ABB RobotStudio station: Proyecto_Final_B2.rspag

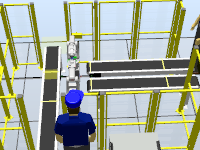
--- station ---
Station Station (saved by RobotStudio 20.4.9280.0)
Controller Controlador3, task T_ROB2: task frame (RAPID world) sits at (-70, -40, 300) mm, rotated rx 0 ry 0 rz -90 deg in the station
Controller Controlador3, task T_ROB1: task frame (RAPID world) sits at (-70, -40, 300) mm, rotated rx 0 ry 0 rz -90 deg in the station
Controller Controlador3
  mechanical unit ROB_1: IRB120_3_58__01, 6 joints, base frame (0, 0, 0) mm
  mechanical unit ROB_2: IRB120_3_58__01_2, 6 joints, base frame (820, 0, 0) mm, rotated rx 0 ry 0 rz 180 deg
Layout (positions relative to the parent item):
  - Conveyor_Cuchara [part]
  - Conveyor_Tenedor [part]
  - Conveyor_Caja [part]
  - Cuchara [part] at (-115.7, -210.79, 5) mm, rotated rx -173.75 ry 0 rz -55.83 deg
  - Tenedor [part] at (40.64, -627.66, 4.91) mm, rotated rx -174.81 ry 0 rz 176.86 deg
  - Logica_Conveyor_Cuchara [smart component]
      signals: DI Start6, DI Start10, DI Start12, DO Sensor_CucharaOK
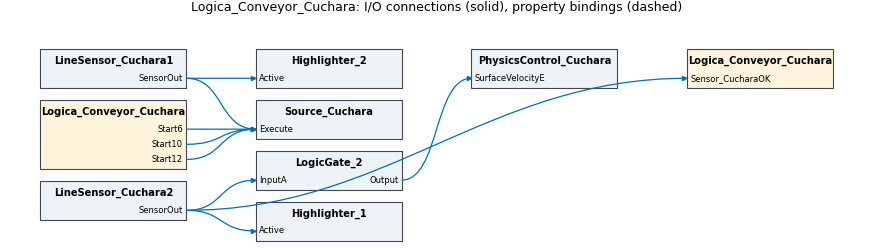
      connections:
        LineSensor_Cuchara1.SensorOut -> Source_Cuchara.Execute
        Logica_Conveyor_Cuchara.Start6 -> Source_Cuchara.Execute
        Logica_Conveyor_Cuchara.Start10 -> Source_Cuchara.Execute
        Logica_Conveyor_Cuchara.Start12 -> Source_Cuchara.Execute
        LineSensor_Cuchara2.SensorOut -> Logica_Conveyor_Cuchara.Sensor_CucharaOK
        LineSensor_Cuchara2.SensorOut -> LogicGate_2.InputA
        LogicGate_2.Output -> PhysicsControl_Cuchara.SurfaceVelocityEnabled
        LineSensor_Cuchara1.SensorOut -> Highlighter_2.Active
        LineSensor_Cuchara2.SensorOut -> Highlighter_1.Active
    - LineSensor_Cuchara1 [smart component, from Components\LineSensor.rslib]
        properties: Start=[1.5 -0.39 0.508]; End=[1.5 -0.11 0.508]; Radius=0.003; SensedPart=(none); SensedPoint=[0 0 0]
      - _sensorPart_ [part]
    - Source_Cuchara [smart component, from Components\Source.rslib]
        properties: Source=Cuchara; Copy=(none); Parent=(none); Position=[1.957 -0.257623 0.5035]; Orientation=[0.154636171726698 0.0188495559215388 0.00453785605518526]; Transient=true; PhysicsBehavior=3
    - LineSensor_Cuchara2 [smart component, from Components\LineSensor.rslib]
        properties: Start=[0.225 -0.39 0.508]; End=[0.225 -0.11 0.508]; Radius=0; SensedPart=(none); SensedPoint=[0.225 -0.212823776245117 0.508]
      - _sensorPart_ [part]
    - PhysicsControl_Cuchara [smart component, from Components\PhysicsControl.rslib]
        properties: Object=Conveyor_Cuchara; Behavior=1; SurfaceVelocity=0.3
    - LogicGate_2 [smart component, from Components\LogicGate.rslib]
        properties: Operator=NOT; Delay=0
    - Highlighter_1 [smart component, from Components\Highlighter.rslib]
        properties: Object=Pilot1; Color=[0 255 0]; Opacity=255
    - Highlighter_2 [smart component, from Components\Highlighter.rslib]
        properties: Object=Pilot2; Color=[0 255 0]; Opacity=255
  - Logica_Conveyor_Tenedor [smart component]
      signals: DI Start6, DI Start10, DI Start12, DO Sensor_TenedorOK
      connections:
        LineSensor_Tenedor.SensorOut -> Source_Tenedor.Execute
        Logica_Conveyor_Tenedor.Start6 -> Source_Tenedor.Execute
        Logica_Conveyor_Tenedor.Start10 -> Source_Tenedor.Execute
        Logica_Conveyor_Tenedor.Start12 -> Source_Tenedor.Execute
        LineSensor_3.SensorOut -> Logica_Conveyor_Tenedor.Sensor_TenedorOK
        LineSensor_3.SensorOut -> LogicGate.InputA
        LogicGate.Output -> PhysicsControl_Tenedor.SurfaceVelocityEnabled
        LineSensor_3.SensorOut -> Highlighter_3.Active
        LineSensor_Tenedor.SensorOut -> Highlighter_4.Active
    - LineSensor_Tenedor [smart component, from Components\LineSensor.rslib]
        properties: Start=[1.5 -0.8 0.508]; End=[1.5 -0.52 0.508]; Radius=0.003; SensedPart=(none); SensedPoint=[0 0 0]
      - _sensorPart_ [part]
    - Source_Tenedor [smart component, from Components\Source.rslib]
        properties: Source=Tenedor; Copy=(none); Parent=(none); Position=[1.957 -0.630695 0.505]; Orientation=[0 0 0]; Transient=true; PhysicsBehavior=3
    - LineSensor_3 [smart component, from Components\LineSensor.rslib]
        properties: Start=[0.228 -0.8 0.508]; End=[0.228 -0.52 0.508]; Radius=0; SensedPart=(none); SensedPoint=[0.227999984741211 -0.719083068847656 0.508]
      - _sensorPart_ [part]
    - PhysicsControl_Tenedor [smart component, from Components\PhysicsControl.rslib]
        properties: Object=Conveyor_Tenedor; Behavior=1; SurfaceVelocity=0.3
    - LogicGate [smart component, from Components\LogicGate.rslib]
        properties: Operator=NOT; Delay=0
    - Highlighter_3 [smart component, from Components\Highlighter.rslib]
        properties: Object=Pilot3; Color=[0 255 0]; Opacity=255
    - Highlighter_4 [smart component, from Components\Highlighter.rslib]
        properties: Object=Pilot4; Color=[0 255 0]; Opacity=255
  - Base_R_Tenedor [part] at (-70, -860, 0) mm
  - Base_R_Cuchara [part] at (-70, -40, 0) mm
  - Caja [part] at (-438.34, 1085.03, 1.58) mm, rotated rx 0 ry 0 rz -1.41 deg
  - Logica_Conveyor_Caja [smart component]
      signals: DI Start6, DI Start10, DI Start12, DO Sensor_CajaOK, DI Rutina
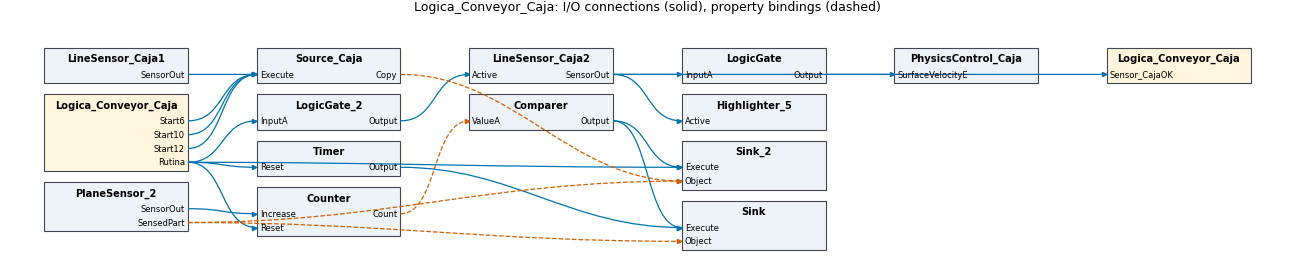
      connections:
        LineSensor_Caja1.SensorOut -> Source_Caja.Execute
        Logica_Conveyor_Caja.Start6 -> Source_Caja.Execute
        Logica_Conveyor_Caja.Start10 -> Source_Caja.Execute
        Logica_Conveyor_Caja.Start12 -> Source_Caja.Execute
        LineSensor_Caja2.SensorOut -> Logica_Conveyor_Caja.Sensor_CajaOK
        LineSensor_Caja2.SensorOut -> LogicGate.InputA
        LogicGate.Output -> PhysicsControl_Caja.SurfaceVelocityEnabled
        Logica_Conveyor_Caja.Rutina -> LogicGate_2.InputA
        LogicGate_2.Output -> LineSensor_Caja2.Active
        Logica_Conveyor_Caja.Rutina -> Sink_2.Execute
        LineSensor_Caja2.SensorOut -> Highlighter_5.Active
        PlaneSensor_2.SensorOut -> Counter.Increase
        Logica_Conveyor_Caja.Rutina -> Counter.Reset
        Comparer.Output -> Sink.Execute
        Comparer.Output -> Sink.Execute
        Timer.Output -> Sink.Execute
        Logica_Conveyor_Caja.Rutina -> Timer.Reset
        PlaneSensor_2.SensedPart => Sink.Object
        Source_Caja.Copy => Sink_2.Object
        Counter.Count => Comparer.ValueA
        PlaneSensor_2.SensedPart => Sink.Object
    - LineSensor_Caja1 [smart component, from Components\LineSensor.rslib]
        properties: Start=[-0.59 -1 0.515]; End=[-0.31 -1 0.515]; Radius=0.005; SensedPart=(none); SensedPoint=[0 0 0]
      - _sensorPart_ [part]
    - Source_Caja [smart component, from Components\Source.rslib]
        properties: Source=Caja2; Copy=(none); Parent=(none); Position=[-0.44646 -1.845404 0.503412]; Orientation=[0 0 0]; Transient=true; PhysicsBehavior=3
    - LineSensor_Caja2 [smart component, from Components\LineSensor.rslib]
        properties: Start=[-0.59 -0.35 0.515]; End=[-0.31 -0.35 0.515]; Radius=0.005; SensedPart=(none); SensedPoint=[-0.546462646484375 -0.35 0.515]
      - _sensorPart_ [part]
    - PhysicsControl_Caja [smart component, from Components\PhysicsControl.rslib]
        properties: Object=Conveyor_Caja; Behavior=1; SurfaceVelocity=0.3
    - LogicGate [smart component, from Components\LogicGate.rslib]
        properties: Operator=NOT; Delay=0
    - PlaneSensor_2 [smart component, from Components\PlaneSensor.rslib]
        properties: Origin=[-0.34 -0.555 0.5545]; Axis1=[-0.21 0 0]; Axis2=[0 0.22 0]; SensedPart=(none)
      - _sensorPart_ [part]
    - LogicGate_2 [smart component, from Components\LogicGate.rslib]
        properties: Operator=NOT; Delay=0
    - Highlighter_5 [smart component, from Components\Highlighter.rslib]
        properties: Object=Pilot5; Color=[0 255 0]; Opacity=255
    - Counter [smart component, from Components\Counter.rslib]
        properties: Count=3
    - Comparer [smart component, from Components\Comparer.rslib]
        properties: ValueA=3; Operator=>=; ValueB=4
    - Sink [smart component, from Components\Sink.rslib]
        properties: Object=(none)
    - Timer [smart component, from Components\Timer.rslib]
        properties: StartTime=10; Interval=10; Repeat=true; CurrentTime=13.728
  - IRB120_3_58__01 [mechanism, from Robots\IRB120_3_58_G_01.rslib] at (-70, -40, 300) mm, rotated rx 0 ry 0 rz -90 deg; joint values [0, 0, 0, 0, 0.5236, 0] (rad or m)
  - IRB120_3_58__01_2 [mechanism, from Robots\IRB120_3_58_G_01.rslib] at (-70, -860, 300) mm, rotated rx 0 ry 0 rz 90 deg; joint values [0, 0, 0, 0, 0.5236, 0] (rad or m)
  - Ventosa_tenedor [smart component, from Libraries\1217c23c-7d3e-48fb-b7d3-d1b2005a3c2bMi_Ventosa.rslib] at (-70, -495.65, 894) mm, rotated rx 180 ry 60 rz -90 deg
      connections:
        Ventosa_tenedor.DI_Coge_Objeto -> ?.Active
        ?.SensorOut -> Attacher.Execute
        Ventosa_tenedor.DI_Coge_Objeto -> LogicGate.InputA
        LogicGate.Output -> Detacher.Execute
        Ventosa_tenedor.DI_Coge_Objeto -> LineSensor.Active
        LineSensor.SensorOut -> Attacher.Execute
        LineSensor.SensedPart => Attacher.Child
        LineSensor.SensedPart => Detacher.Child
    - Attacher [smart component, from Components\Attacher.rslib]
        properties: Parent=Ventosa; Flange=0; Child=(none); Mount=false; Offset=[0 0 0]; Orientation=[0 0 0]
    - Detacher [smart component, from Components\Detacher.rslib]
        properties: Child=(none); KeepPosition=true
    - Ventosa [mechanism, from Libraries\1217c23c-7d3e-48fb-b7d3-d1b2005a3c2bMi_Ventosa.rslib] at (0, 0, 0) mm
    - LogicGate [smart component, from Components\LogicGate.rslib]
        properties: Operator=NOT; Delay=0
    - LineSensor [smart component, from Components\LineSensor.rslib]
        properties: Start=[5.20373137080643E-08 6.3539233263743E-08 0.0549999072719709]; End=[5.18797551862793E-08 6.35131238713171E-08 0.062499907271971]; Radius=0; SensedPart=(none); SensedPoint=[-0.419999938964844 -0.519800048828125 0.560922058105469]
      - _sensorPart_ [part]
    - Indicador [part, from Libraries\1217c23c-7d3e-48fb-b7d3-d1b2005a3c2bMi_Ventosa.rslib] at (-4.38, 0, 0) mm
  - Ventosa_cuchara [smart component, from Libraries\1217c23c-7d3e-48fb-b7d3-d1b2005a3c2bMi_Ventosa.rslib] at (-70, -404.35, 894) mm, rotated rx 180 ry 60 rz 90 deg
      connections:
        Ventosa_cuchara.DI_Coge_Objeto -> ?.Active
        ?.SensorOut -> Attacher.Execute
        Ventosa_cuchara.DI_Coge_Objeto -> LogicGate.InputA
        LogicGate.Output -> Detacher.Execute
        Ventosa_cuchara.DI_Coge_Objeto -> LineSensor.Active
        LineSensor.SensorOut -> Attacher.Execute
        LineSensor.SensedPart => Attacher.Child
        LineSensor.SensedPart => Detacher.Child
    - Attacher [smart component, from Components\Attacher.rslib]
        properties: Parent=Ventosa; Flange=0; Child=(none); Mount=false; Offset=[0 0 0]; Orientation=[0 0 0]
    - Detacher [smart component, from Components\Detacher.rslib]
        properties: Child=(none); KeepPosition=true
    - Ventosa [mechanism, from Libraries\1217c23c-7d3e-48fb-b7d3-d1b2005a3c2bMi_Ventosa.rslib] at (0, 0, 0) mm
    - LogicGate [smart component, from Components\LogicGate.rslib]
        properties: Operator=NOT; Delay=0
    - LineSensor [smart component, from Components\LineSensor.rslib]
        properties: Start=[0 0 0.055]; End=[-1.13103603149867E-08 -1.19271307830182E-08 0.0619999031141458]; Radius=0; SensedPart=(none); SensedPoint=[-0.419999969482422 -0.376149993896484 0.56155517578125]
      - _sensorPart_ [part]
    - Indicador [part, from Libraries\1217c23c-7d3e-48fb-b7d3-d1b2005a3c2bMi_Ventosa.rslib] at (-4.38, 0, 0) mm
  - Fence [graphiccomponentgroup]
    - Segment 1 [part]
    - Segment 2 [part]
    - Segment 3 [part]
    - Segment 4 [part]
    - Segment 5 [part]
  - Fence [graphiccomponentgroup]
    - Segment 1 [part]
    - Segment 2 [part]
    - Segment 3 [part]
    - Segment 4 [part]
    - Segment 5 [part]
  - Fence [graphiccomponentgroup]
    - Segment 1 [part]
    - Segment 2 [part]
    - Segment 3 [part]
    - Segment 4 [part]
    - Segment 5 [part]
    - Segment 6 [part]
  - IRC5_Control-Module [part, from Equipment\IRC5_Control-Module.rslib] at (800, -2180, 100) mm, rotated rx 90 ry 0 rz 0 deg
  - PlaneSensor [smart component, from Components\PlaneSensor.rslib]
      properties: Origin=[-0.7 0.32 0.3]; Axis1=[0.5 0 0]; Axis2=[0 0.5 0]; SensedPart=(none)
    - _sensorPart_ [part]
  - Sink [smart component, from Components\Sink.rslib]
      properties: Object=(none)
  - Man2 [part, from Libraries\b1fed280-7d32-4964-bca3-7f8177a599d8man2.rslib] at (2300, 0, 0) mm, rotated rx 0 ry 0 rz 180 deg
  - Man2_2 [part, from Libraries\b1fed280-7d32-4964-bca3-7f8177a599d8man2.rslib] at (-100, -2200, 0) mm, rotated rx 0 ry 0 rz 90 deg
  - Placa1 [part] at (200, -410, 400) mm
  - Placa3 [part] at (-200, -620, -50) mm
  - Placa2 [part]
  - Placa4 [part]
  - Placa5 [part]
  - Pilot5 [part]
  - Pilot1 [part]
  - Pilot2 [part]
  - Pilot4 [part]
  - Pilot3 [part]
  - Placa6 [part]
  - Pilot_r_tenedor [part] at (0, 14.72, 0) mm
  - Pilot_r_cuchara [part] at (0, -7.35, 0) mm
  - Highlighter_r_cuchara [smart component, from Components\Highlighter.rslib]
      properties: Object=Pilot_r_cuchara; Color=[0 255 0]; Opacity=255
  - Highlighter_r_tenedor [smart component, from Components\Highlighter.rslib]
      properties: Object=Pilot_r_tenedor; Color=[0 255 0]; Opacity=255
  - Caja2 [part] at (-14.34, -14695.99, 1.59) mm, rotated rx 0 ry 0 rz 5.75 deg
Attachment: Ventosa_tenedor is attached to IRB120_3_58__01_2 / Link6
Attachment: Ventosa_cuchara is attached to IRB120_3_58__01 / Link6
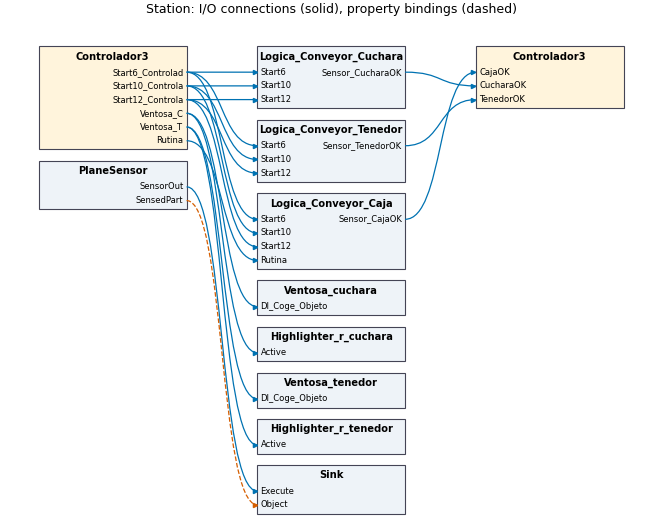
Station logic (signal -> signal, property => property):
  Controlador3.Start6_Controlador -> Logica_Conveyor_Caja.Start6
  Controlador3.Start10_Controlador -> Logica_Conveyor_Caja.Start10
  Controlador3.Start12_Controlador -> Logica_Conveyor_Caja.Start12
  Controlador3.Start6_Controlador -> Logica_Conveyor_Cuchara.Start6
  Controlador3.Start10_Controlador -> Logica_Conveyor_Cuchara.Start10
  Controlador3.Start12_Controlador -> Logica_Conveyor_Cuchara.Start12
  Controlador3.Start6_Controlador -> Logica_Conveyor_Tenedor.Start6
  Controlador3.Start10_Controlador -> Logica_Conveyor_Tenedor.Start10
  Controlador3.Start12_Controlador -> Logica_Conveyor_Tenedor.Start12
  Logica_Conveyor_Caja.Sensor_CajaOK -> Controlador3.CajaOK
  Logica_Conveyor_Cuchara.Sensor_CucharaOK -> Controlador3.CucharaOK
  Logica_Conveyor_Tenedor.Sensor_TenedorOK -> Controlador3.TenedorOK
  Controlador3.Ventosa_C -> Ventosa_cuchara.DI_Coge_Objeto
  Controlador3.Ventosa_T -> Ventosa_tenedor.DI_Coge_Objeto
  Controlador3.Rutina -> Logica_Conveyor_Caja.Rutina
  PlaneSensor.SensorOut -> Sink.Execute
  Controlador3.Ventosa_C -> Highlighter_r_cuchara.Active
  Controlador3.Ventosa_T -> Highlighter_r_tenedor.Active
  PlaneSensor.SensedPart => Sink.Object

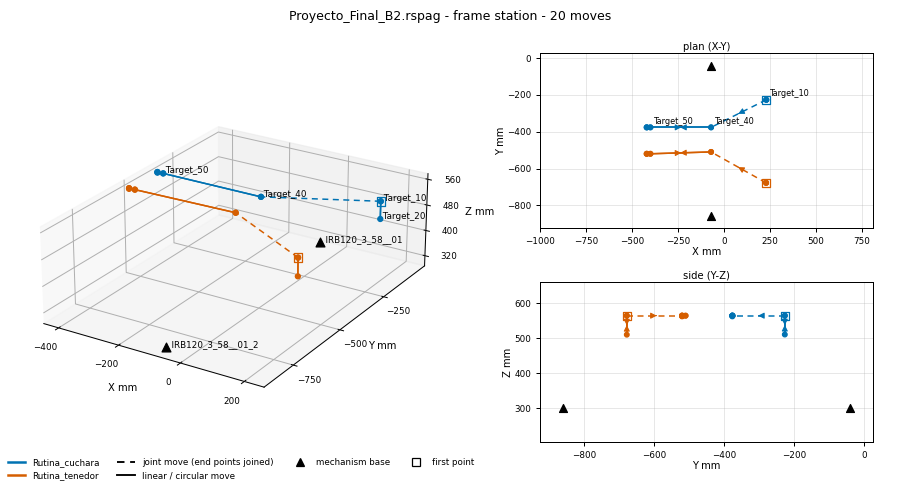
[picture p0: tool path of Proyecto_Final_B2.rspag in frame station, 20 of 20 moves have a stored position in this frame; points joined in program order, loops and branches not executed]
--- Backups/Controlador3/RAPID/TASK1/PROGMOD/CalibData.mod ---
MODULE CalibData
    PERS tooldata TCP_Ventosa:=[TRUE,[[0,0,60],[1,0,0,0]],[0.1,[0,0,1],[1,0,0,0],0,0,0]];
    TASK PERS wobjdata Workobject_1:=[FALSE,TRUE,"",[[210,270,200],[1,0,0,0]],[[0,0,0],[1,0,0,0]]];
    PERS tooldata Tooldata_1:=[TRUE,[[0,0,60],[1,0,0,0]],[0.1,[0,0,1],[1,0,0,0],0,0,0]];
ENDMODULE

--- Backups/Controlador3/RAPID/TASK1/PROGMOD/Module1.mod ---
MODULE Module1
    CONST robtarget Target_10:=[[-23.679995733,30.000024272,64.999939178],[0.000000004,0,1,0.000000007],[0,0,0,0],[9E+09,9E+09,9E+09,9E+09,9E+09,9E+09]];
    CONST robtarget Target_20:=[[-23.68,30,11.2],[0,0,1,0],[0,0,0,0],[9E+09,9E+09,9E+09,9E+09,9E+09,9E+09]];
    CONST robtarget Target_30:=[[-23.679995733,30.000024272,64.999939178],[0.000000004,0,1,0.000000007],[0,0,0,0],[9E+09,9E+09,9E+09,9E+09,9E+09,9E+09]];
    CONST robtarget Target_40:=[[126.149990693,-270.119999999,64.999933168],[0.000000011,0.486182918,0.873857065,0.000000019],[-1,0,0,0],[9E+09,9E+09,9E+09,9E+09,9E+09,9E+09]];
    CONST robtarget Target_50:=[[126.149993351,-600.000025877,64.999935931],[0.000000004,0.4861829,0.873857075,-0.000000015],[-1,-1,0,0],[9E+09,9E+09,9E+09,9E+09,9E+09,9E+09]];
    CONST robtarget Target_60:=[[126.15,-620,65],[0,0.707106781,0.707106781,0],[-1,-1,0,0],[9E+09,9E+09,9E+09,9E+09,9E+09,9E+09]];
    CONST robtarget Target_70:=[[126.15,-620,63],[0,0.707106781,0.707106781,0],[-1,-1,0,0],[9E+09,9E+09,9E+09,9E+09,9E+09,9E+09]];
    VAR num contador:=0;
    !***********************************************************
    !
    ! Módulo:  Module1
    !
    ! Descripción:
    !   <Introduzca la descripción aquí>
    !
    ! Autor: Admin
    !
    ! Versión: 1.0
    !
    !***********************************************************


    !***********************************************************
    !
    ! Procedimiento Main
    !
    !   Este es el punto de entrada de su programa
    !
    !***********************************************************
    !Declaración de variables de interrupción

    VAR intnum int_buttonStopDI;                           !intnum comando que identifica interrupcion de parada de emergencia.

    PROC main()
        !Añada aquí su código
        setDO Start6_Controlador,0;
        setDO Start10_Controlador,0;
        setDO Start12_Controlador,0;
        SetDO Ventosa_C,0;
        SetDO Rutina,0;
        ciclo_inicio_cuchara:
        IF cubiertos_6=high THEN
            IDelete int_buttonStopDI;                          !Cancela interrupcion, necesario cuando el ciclo se repite.
            CONNECT int_buttonStopDI WITH parada_emergencia;   !Se conecta la rutina TRAP con la interrupicion parada_emergencia
            iSignalDI Stop_button, 1, int_buttonStopDI;         !Se asocia buttonStop con la interrupcion parada_emergencia
            setDO Start6_Controlador,1;
            !setDO Start6_Controlador, 0;
            contador:=6;
            Rutina_cuchara;
            SetDO Rutina,1;
            WaitTime 1.5;
            SetDO Rutina,0;
        ELSEIF cubiertos_10=high THEN
            IDelete int_buttonStopDI;                          !Cancela interrupcion, necesario cuando el ciclo se repite.
            CONNECT int_buttonStopDI WITH parada_emergencia;   !Se conecta la rutina TRAP con la interrupicion parada_emergencia
            iSignalDI Stop_button, 1, int_buttonStopDI;         !Se asocia buttonStop con la interrupcion parada_emergencia
            setDO Start10_Controlador,1;
            !setDO Start10_Controlador, 0;
            contador:=10;
            Rutina_cuchara;
            SetDO Rutina,1;
            WaitTime 1.5;
            SetDO Rutina,0;
        ELSEIF cubiertos_12=high THEN
            IDelete int_buttonStopDI;                          !Cancela interrupcion, necesario cuando el ciclo se repite.
            CONNECT int_buttonStopDI WITH parada_emergencia;   !Se conecta la rutina TRAP con la interrupicion parada_emergencia
            iSignalDI Stop_button, 1, int_buttonStopDI;         !Se asocia buttonStop con la interrupcion parada_emergencia
            setDO Start12_Controlador,1;
            !setDO Start12_Controlador, 0;
            contador:=12;
            Rutina_cuchara;
            SetDO Rutina,1;
            WaitTime 1.5;
            SetDO Rutina,0;
        ELSE
            GOTO ciclo_inicio_cuchara;
        ENDIF
    ENDPROC
    PROC Rutina_cuchara()
        WHILE contador>0 DO
            WaitDI CajaOK,1;
            WaitDI CucharaOK,1;
            WaitDI TenedorOK,1;
            MoveJ Target_10,v600,z10,TCP_Ventosa\WObj:=Workobject_1;
            MoveL Target_20,v50,z1,TCP_Ventosa\WObj:=Workobject_1;
            SetDO Ventosa_C,1;
            WaitTime 1;
            MoveL Target_30,v150,z1,TCP_Ventosa\WObj:=Workobject_1;
            MoveJ Target_40,v600,z10,TCP_Ventosa\WObj:=Workobject_1;
            MoveL Target_50,v300,z1,TCP_Ventosa\WObj:=Workobject_1;
            MoveL Target_60,v300,z1,TCP_Ventosa\WObj:=Workobject_1;
            MoveL Target_70,v10,fine,Tooldata_1\WObj:=Workobject_1;
            SetDO Ventosa_C,0;
            WaitTime 1;
            MoveL Target_60,v300,z1,TCP_Ventosa\WObj:=Workobject_1;
            MoveL Target_50,v300,z1,TCP_Ventosa\WObj:=Workobject_1;
            MoveL Target_40,v300,z1,TCP_Ventosa\WObj:=Workobject_1;
            contador:=contador-1;
            IF contador=0 THEN
                IF cubiertos_6=high THEN
                   contador:=6;
                   SetDO Rutina,1;
                   WaitTime 1.5;
                   SetDO Rutina,0;
                ELSEIF cubiertos_10=high THEN
                   contador:=10;
                   SetDO Rutina,1;
                   WaitTime 1.5;
                   SetDO Rutina,0;
                ELSEIF cubiertos_12=high THEN
                   contador:=12;
                   SetDO Rutina,1;
                   WaitTime 1.5;
                   SetDO Rutina,0;
                ENDIF
            ENDIF
        ENDWHILE
    ENDPROC

    TRAP parada_emergencia                              !Interrupcion parada_emergencia
        StopMove;                                       !Detiene movimento de robot
        SetDO Rutina,0;
        !IF buttonStop=low THEN
        !    StartMove;
        !ELSE
        !    parada_emergencia:
        !ENDIF
        WHILE Stop_button = high DO                      !Mientras siga activo pulsador buttonStop, el programa seguirá detenido
        ENDWHILE
        StartMove;                                      !Si se desactiva pulsador buttonStop, el programa continua donde quedó.
    ENDTRAP
ENDMODULE

--- Backups/Controlador3/RAPID/TASK1/SYSMOD/LINKEDM.sys ---
%%%
  VERSION:1
  LANGUAGE:ENGLISH
%%%

MODULE LINKEDM (SYSMODULE)

! FOLLOWER
!     Name of electronically linked follower axis used by operator at teach pendent.
      PERS string l_f_axis_name{5}       :=  ["",  "", "", "", ""];

!     Name of the mechanical unit for follower axis.
      PERS string l_f_mecunt_n{5}  :=  ["", "", "", "", ""];

!     Linked follower axis number in the mechanical unit (first axis in mech. unit is number 1).
      PERS num l_f_axis_no{5}      :=  [0,          0,   0,  0,  0];

! MASTER
!     Name of the mechanical unit for linked master axis.
      PERS string l_m_mecunt_n{5} :=  ["", "", "", "", ""];

!     Linked master axis number in the mechanical unit (first axis in mech. unit is number 1).
!     See axis number table in documentation for different master mechanical units.
      PERS num l_m_axis_no{5}     :=  [0,  0,  0,  0,  0];

! POSITION OFFSET
!     The increase of the allowed offset position between the master and follower
!     positions, used when starting AUTO mode. As soon as the offset is decreased
!     the old configurated parameter is used.
!     Example: 3 => the configurated value of allowed offset is increased 3 times.
      PERS num offset_ratio{5}       :=  [10,  10,   10,  10,  10];

! SPEED RATIO
!     Speed_ratio used in AUTO and JOG modes [ very_slow   slow    normal    fast]
!     Value 1 = max allowed manual speed.
      CONST num speed_ratio {20}      := [0.01, 0.01, 0.01, 0.01, 0.01,
                                          0.05, 0.05, 0.05, 0.05, 0.05,
                                          0.20, 0.20, 0.20, 0.20, 0.20,
                                          1.00, 1.00, 1.00, 1.00, 1.00];

! STEP SIZE
!     Displacement position used in JOG mode for each activation of positive or
!     negative movement.                  [very_short    short   normal   long]
!     Unit degees or meter.
      CONST num displacement {20}     := [0.001, 0.001, 0.001, 0.001, 0.001,
                                          0.005, 0.005, 0.005, 0.005, 0.005,
                                          0.020, 0.020, 0.020, 0.020, 0.020,
                                          0.100, 0.100, 0.100, 0.100, 0.100];


!-------------------------------------------------------------
 PROC Linked_m ()
      Linked_m_exe ;
 ENDPROC
ENDMODULE

--- Backups/Controlador3/RAPID/TASK2/PROGMOD/CalibData.mod ---
MODULE CalibData
    PERS tooldata TCP_Ventosa:=[TRUE,[[0,0,60],[1,0,0,0]],[0.1,[0,0,1],[1,0,0,0],0,0,0]];
    TASK PERS wobjdata Workobject_2:=[FALSE,TRUE,"",[[620,270,200],[1,0,0,0]],[[0,0,0],[1,0,0,0]]];
ENDMODULE

--- Backups/Controlador3/RAPID/TASK2/PROGMOD/Module1.mod ---
MODULE Module1
    CONST robtarget Target_10:=[[17.680006378,29.000003785,64.999943406],[-0.000000006,1,0,0.000000004],[-1,0,-1,0],[9E+09,9E+09,9E+09,9E+09,9E+09,9E+09]];
    CONST robtarget Target_20:=[[17.68,29,10.7],[0,1,0,0],[-1,-1,-1,0],[9E+09,9E+09,9E+09,9E+09,9E+09,9E+09]];
    CONST robtarget Target_30:=[[17.680006378,29.000003785,64.999943406],[-0.000000006,1,0,0.000000004],[-1,0,-1,0],[9E+09,9E+09,9E+09,9E+09,9E+09,9E+09]];
    CONST robtarget Target_40:=[[-150.200005115,-270.140000008,64.999941394],[-0.000000007,0.871855665,0.489762902,0.000000004],[0,0,-1,0],[9E+09,9E+09,9E+09,9E+09,9E+09,9E+09]];
    CONST robtarget Target_50:=[[-140.200013899,-600.000004341,64.999949592],[0.000000013,0.871855673,0.489762887,0.000000004],[0,-1,-1,0],[9E+09,9E+09,9E+09,9E+09,9E+09,9E+09]];
    CONST robtarget Target_60:=[[-140.2,-620,65],[0,0.707106781,0.707106781,0],[0,-1,-1,0],[9E+09,9E+09,9E+09,9E+09,9E+09,9E+09]];
    CONST robtarget Target_70:=[[-140.2,-620,63],[0,0.707106781,0.707106781,0],[0,0,-1,0],[9E+09,9E+09,9E+09,9E+09,9E+09,9E+09]];
    VAR num contador:=0;
    !***********************************************************
    !
    ! Módulo:  Module1
    !
    ! Descripción:
    !   <Introduzca la descripción aquí>
    !
    ! Autor: Admin
    !
    ! Versión: 1.0
    !
    !***********************************************************


    !***********************************************************
    !
    ! Procedimiento Main
    !
    !   Este es el punto de entrada de su programa
    !
    !***********************************************************
    !Declaración de variables de interrupción

    VAR intnum int_buttonStopDI;                           !intnum comando que identifica interrupcion de parada de emergencia.

    PROC main()
        !Añada aquí su código
        setDO Start6_Controlador,0;
        setDO Start10_Controlador,0;
        setDO Start12_Controlador,0;
        SetDO Rutina,0;
        SetDO Ventosa_T,0;
        ciclo_inicio_tenedor:
        IF cubiertos_6=high THEN
            IDelete int_buttonStopDI;                          !Cancela interrupcion, necesario cuando el ciclo se repite.
            CONNECT int_buttonStopDI WITH parada_emergencia;   !Se conecta la rutina TRAP con la interrupicion parada_emergencia
            iSignalDI Stop_button, 1, int_buttonStopDI;         !Se asocia buttonStop con la interrupcion parada_emergencia
            setDO Start6_Controlador,1;
            !setDO Start6_Controlador, 0;
            contador:=6;
            Rutina_tenedor;
            SetDO Rutina,1;
            WaitTime 1.5;
            SetDO Rutina,0;
        ELSEIF cubiertos_10=high THEN
            IDelete int_buttonStopDI;                          !Cancela interrupcion, necesario cuando el ciclo se repite.
            CONNECT int_buttonStopDI WITH parada_emergencia;   !Se conecta la rutina TRAP con la interrupicion parada_emergencia
            iSignalDI Stop_button, 1, int_buttonStopDI;         !Se asocia buttonStop con la interrupcion parada_emergencia
            setDO Start10_Controlador,1;
            !setDO Start10_Controlador, 0;
            contador:=10;
            Rutina_tenedor;
            SetDO Rutina,1;
            WaitTime 1.5;
            SetDO Rutina,0;
        ELSEIF cubiertos_12=high THEN
            IDelete int_buttonStopDI;                          !Cancela interrupcion, necesario cuando el ciclo se repite.
            CONNECT int_buttonStopDI WITH parada_emergencia;   !Se conecta la rutina TRAP con la interrupicion parada_emergencia
            iSignalDI Stop_button, 1, int_buttonStopDI;         !Se asocia buttonStop con la interrupcion parada_emergencia
            setDO Start12_Controlador,1;
            !setDO Start12_Controlador, 0;
            contador:=12;
            Rutina_tenedor;
            SetDO Rutina,1;
            WaitTime 1.5;
            SetDO Rutina,0;
        ELSE
            GOTO ciclo_inicio_tenedor;
        ENDIF
    ENDPROC
    PROC Rutina_tenedor()
        WHILE contador>0 DO
            WaitDI CajaOK,1;
            WaitDI CucharaOK,1;
            WaitDI TenedorOK,1;
            MoveJ Target_10,v600,z10,TCP_Ventosa\WObj:=Workobject_2;
            MoveL Target_20,v50,z1,TCP_Ventosa\WObj:=Workobject_2;
            SetDO Ventosa_T,1;
            WaitTime 1;
            MoveL Target_30,v150,z1,TCP_Ventosa\WObj:=Workobject_2;
            MoveJ Target_40,v600,z10,TCP_Ventosa\WObj:=Workobject_2;
            MoveL Target_50,v300,z1,TCP_Ventosa\WObj:=Workobject_2;
            MoveL Target_60,v300,z1,TCP_Ventosa\WObj:=Workobject_2;
            MoveL Target_70,v10,fine,TCP_Ventosa\WObj:=Workobject_2;
            SetDO Ventosa_T,0;
            WaitTime 1;
            MoveL Target_60,v300,z1,TCP_Ventosa\WObj:=Workobject_2;
            MoveL Target_50,v300,z1,TCP_Ventosa\WObj:=Workobject_2;
            MoveL Target_40,v300,z1,TCP_Ventosa\WObj:=Workobject_2;
            contador:=contador-1;
            IF contador=0 THEN
                IF cubiertos_6=high THEN
                   contador:=6;
                   SetDO Rutina,1;
                   WaitTime 1.5;
                   SetDO Rutina,0;
                ELSEIF cubiertos_10=high THEN
                   contador:=10;
                   SetDO Rutina,1;
                   WaitTime 1.5;
                   SetDO Rutina,0;
                ELSEIF cubiertos_12=high THEN
                   contador:=12;
                   SetDO Rutina,1;
                   WaitTime 1.5;
                   SetDO Rutina,0;
                ENDIF
            ENDIF
        ENDWHILE
    ENDPROC

   TRAP parada_emergencia                              !Interrupcion parada_emergencia
        StopMove;                                       !Detiene movimento de robot
        SetDO Rutina,0;
        !IF buttonStop=low THEN
        !    StartMove;
        !ELSE
        !    parada_emergencia:
        !ENDIF
        WHILE Stop_button = high DO                      !Mientras siga activo pulsador buttonStop, el programa seguirá detenido
        ENDWHILE
        StartMove;                                      !Si se desactiva pulsador buttonStop, el programa continua donde quedó.
    ENDTRAP
ENDMODULE

--- Backups/Controlador3/SYSPAR/EIO.cfg ---
EIO:CFG_1.0:6:1::
#
EIO_SIGNAL:

      -Name "cubiertos_6" -SignalType "DI"\
      -Label "Esta senal undica que el numero de cubiertos que cogera el robot, seran 6"\
      -Access "All"

      -Name "cubiertos_10" -SignalType "DI"\
      -Label "Esta senal undica que el numero de cubiertos que cogera el robot, seran 10"\
      -Access "All"

      -Name "cubiertos_12" -SignalType "DI"\
      -Label "Esta senal undica que el numero de cubiertos que cogera el robot, seran 12"\
      -Access "All"

      -Name "Start6_Controlador" -SignalType "DO"\
      -Label "Senal de salida que inicia la rutina de 6 cubiertos" -Access "All"

      -Name "Start10_Controlador" -SignalType "DO"\
      -Label "Senal de salida que inicia la rutina de 10 cubiertos"\
      -Access "All"

      -Name "Start12_Controlador" -SignalType "DO"\
      -Label "Senal de salida que inicia la rutina de 12 cubiertos"\
      -Access "All"

      -Name "CajaOK" -SignalType "DI"\
      -Label "Esta senal indica que la caja ya esta en su posicion para recibir cucharas"\
      -Access "All"

      -Name "CucharaOK" -SignalType "DI"\
      -Label "Esta senal indica que la cuchara ya esta en su posicion para ser tomada por la v"\
      -Access "All"

      -Name "TenedorOK" -SignalType "DI"\
      -Label "Esta senal indica que el tenedor ya esta en su posicion para ser tomada por la v"\
      -Access "All"

      -Name "Ventosa_C" -SignalType "DO"\
      -Label "Senal que produce que la ventosa coja o suelte la cuchara "\
      -Access "All"

      -Name "Ventosa_T" -SignalType "DO"\
      -Label "Senal que produce que la ventosa coja o suelte el tenedor "\
      -Access "All"

      -Name "Rutina" -SignalType "DO"\
      -Label "Senal necesaria para activar o desactivar el enabled de PhysicsControl de la ban"\
      -Access "All"

      -Name "Stop_button" -SignalType "DI"\
      -Label "senal del boton parada de emergencia que detiene operacion"\
      -Access "All"
